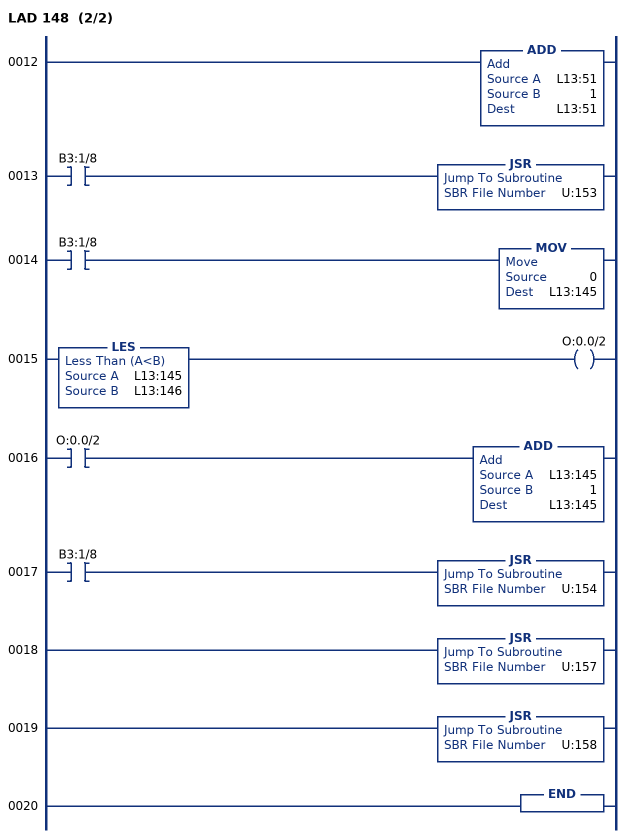
% Rung: 12 %
SOR ADD L13:51 1 L13:51 EOR
% Rung: 13 %
SOR XIC B3:1/8 JSR U:153 EOR
% Rung: 14 %
SOR XIC B3:1/8 MOV 0 L13:145 EOR
% Rung: 15 %
SOR LES L13:145 L13:146 OTE O:0.0/2 EOR
% Rung: 16 %
SOR XIC O:0.0/2 ADD L13:145 1 L13:145 EOR
% Rung: 17 %
SOR XIC B3:1/8 JSR U:154 EOR
% Rung: 18 %
SOR JSR U:157 EOR
% Rung: 19 %
SOR JSR U:158 EOR
% Rung: 20 %
SOR END EOR

LADDER 149
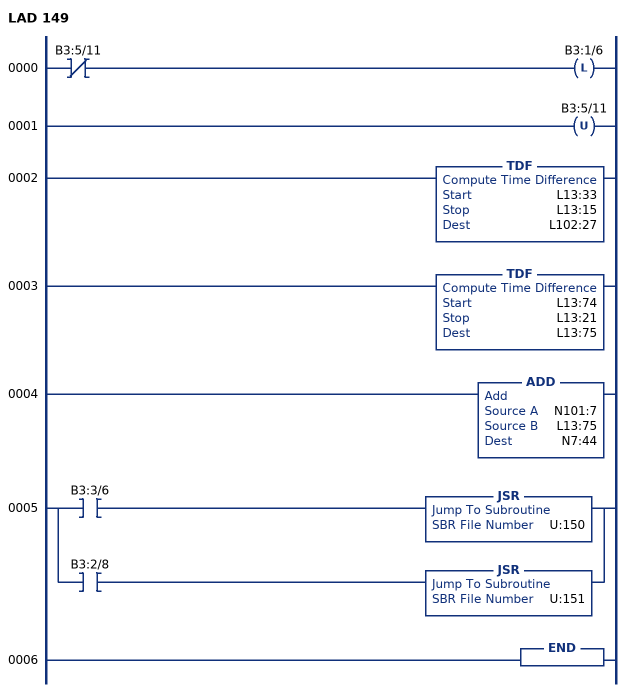
% Rung: 0 %
SOR XIO B3:5/11 OTL B3:1/6 EOR
% Rung: 1 %
SOR OTU B3:5/11 EOR
% Rung: 2 %
SOR TDF L13:33 L13:15 L102:27 EOR
% Rung: 3 %
SOR TDF L13:74 L13:21 L13:75 EOR
% Rung: 4 %
SOR ADD N101:7 L13:75 N7:44 EOR
% Rung: 5 %
SOR BST XIC B3:3/6 JSR U:150 NXB XIC B3:2/8 JSR U:151 BND EOR
% Rung: 6 %
SOR END EOR

LADDER 150
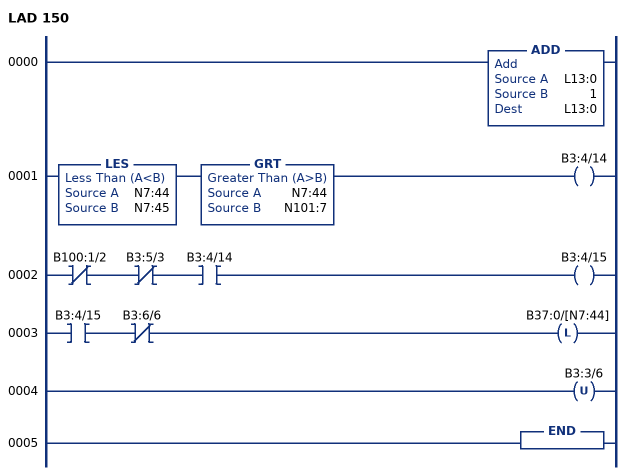
% Rung: 0 %
SOR ADD L13:0 1 L13:0 EOR
% Rung: 1 %
SOR LES N7:44 N7:45 GRT N7:44 N101:7 OTE B3:4/14 EOR
% Rung: 2 %
SOR XIO B100:1/2 XIO B3:5/3 XIC B3:4/14 OTE B3:4/15 EOR
% Rung: 3 %
SOR XIC B3:4/15 XIO B3:6/6 OTL B37:0/[N7:44] EOR
% Rung: 4 %
SOR OTU B3:3/6 EOR
% Rung: 5 %
SOR END EOR

LADDER 151
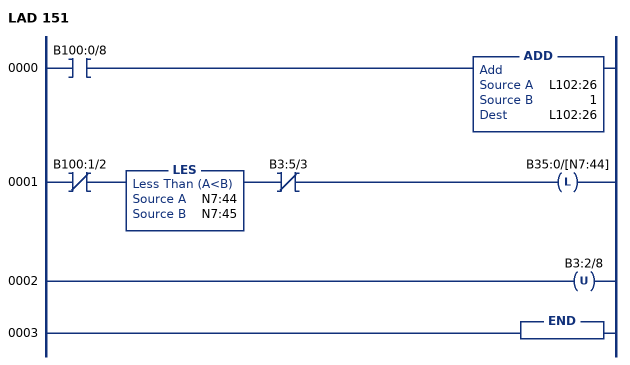
% Rung: 0 %
SOR XIC B100:0/8 ADD L102:26 1 L102:26 EOR
% Rung: 1 %
SOR XIO B100:1/2 LES N7:44 N7:45 XIO B3:5/3 OTL B35:0/[N7:44] EOR
% Rung: 2 %
SOR OTU B3:2/8 EOR
% Rung: 3 %
SOR END EOR

LADDER 152
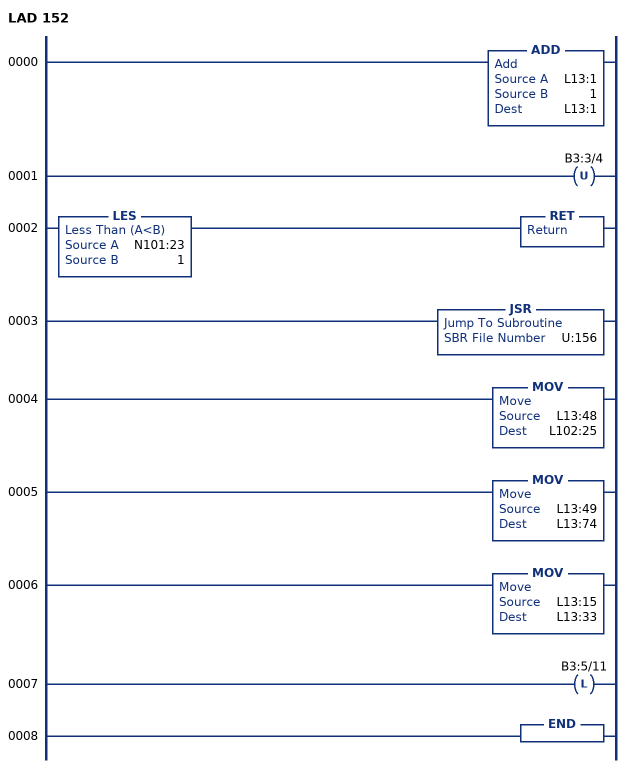
% Rung: 0 %
SOR ADD L13:1 1 L13:1 EOR
% Rung: 1 %
SOR OTU B3:3/4 EOR
% Rung: 2 %
SOR LES N101:23 1 RET EOR
% Rung: 3 %
SOR JSR U:156 EOR
% Rung: 4 %
SOR MOV L13:48 L102:25 EOR
% Rung: 5 %
SOR MOV L13:49 L13:74 EOR
% Rung: 6 %
SOR MOV L13:15 L13:33 EOR
% Rung: 7 %
SOR OTL B3:5/11 EOR
% Rung: 8 %
SOR END EOR

LADDER 153
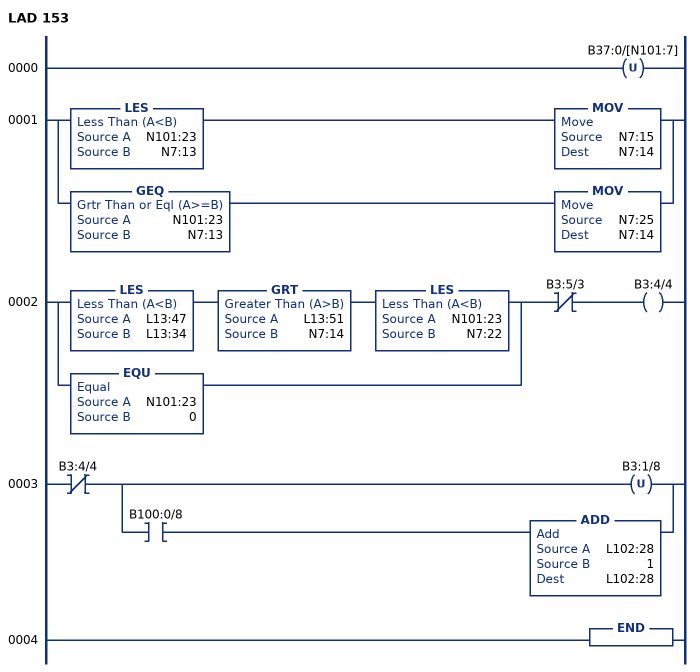
% Rung: 0 %
SOR OTU B37:0/[N101:7] EOR
% Rung: 1 %
SOR BST LES N101:23 N7:13 MOV N7:15 N7:14 NXB GEQ N101:23 N7:13 MOV N7:25 N7:14 BND EOR
% Rung: 2 %
SOR BST LES L13:47 L13:34 GRT L13:51 N7:14 LES N101:23 N7:22 NXB EQU N101:23 0 BND XIO B3:5/3 OTE B3:4/4 EOR
% Rung: 3 %
SOR XIO B3:4/4 BST OTU B3:1/8 NXB XIC B100:0/8 ADD L102:28 1 L102:28 BND EOR
% Rung: 4 %
SOR END EOR

LADDER 154
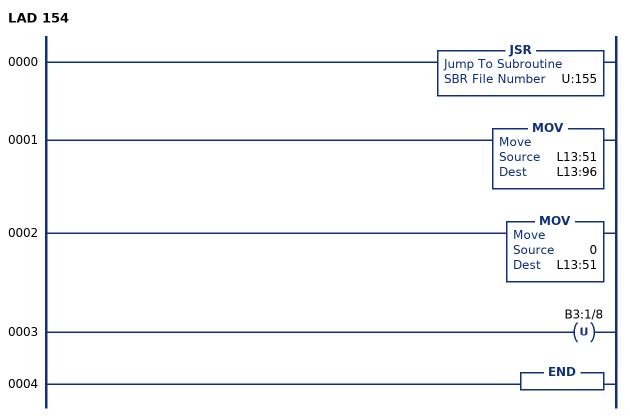
% Rung: 0 %
SOR JSR U:155 EOR
% Rung: 1 %
SOR MOV L13:51 L13:96 EOR
% Rung: 2 %
SOR MOV 0 L13:51 EOR
% Rung: 3 %
SOR OTU B3:1/8 EOR
% Rung: 4 %
SOR END EOR

LADDER 155
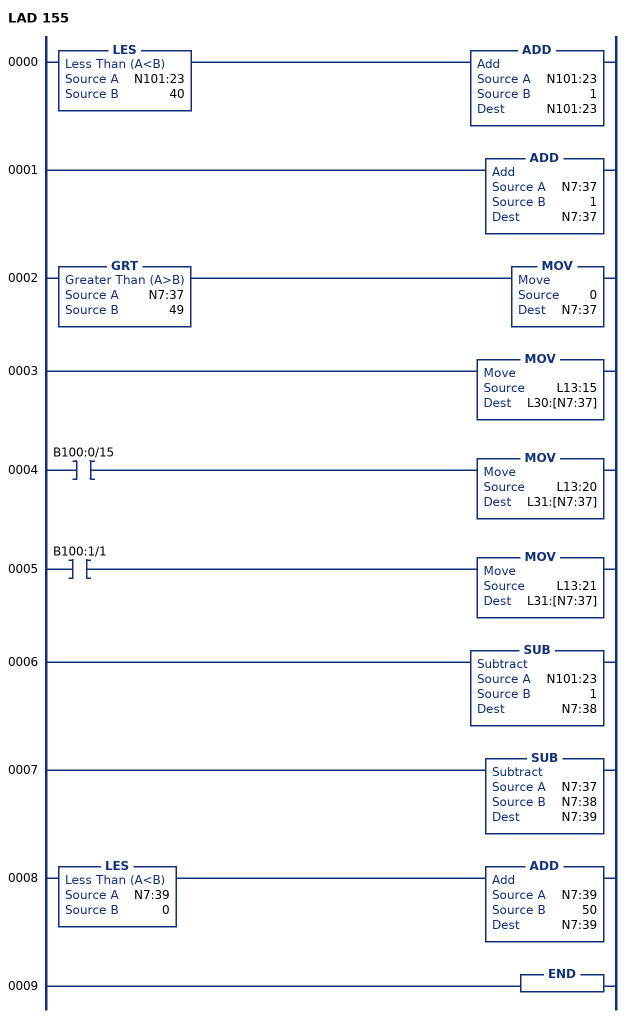
% Rung: 0 %
SOR LES N101:23 40 ADD N101:23 1 N101:23 EOR
% Rung: 1 %
SOR ADD N7:37 1 N7:37 EOR
% Rung: 2 %
SOR GRT N7:37 49 MOV 0 N7:37 EOR
% Rung: 3 %
SOR MOV L13:15 L30:[N7:37] EOR
% Rung: 4 %
SOR XIC B100:0/15 MOV L13:20 L31:[N7:37] EOR
% Rung: 5 %
SOR XIC B100:1/1 MOV L13:21 L31:[N7:37] EOR
% Rung: 6 %
SOR SUB N101:23 1 N7:38 EOR
% Rung: 7 %
SOR SUB N7:37 N7:38 N7:39 EOR
% Rung: 8 %
SOR LES N7:39 0 ADD N7:39 50 N7:39 EOR
% Rung: 9 %
SOR END EOR

LADDER 156
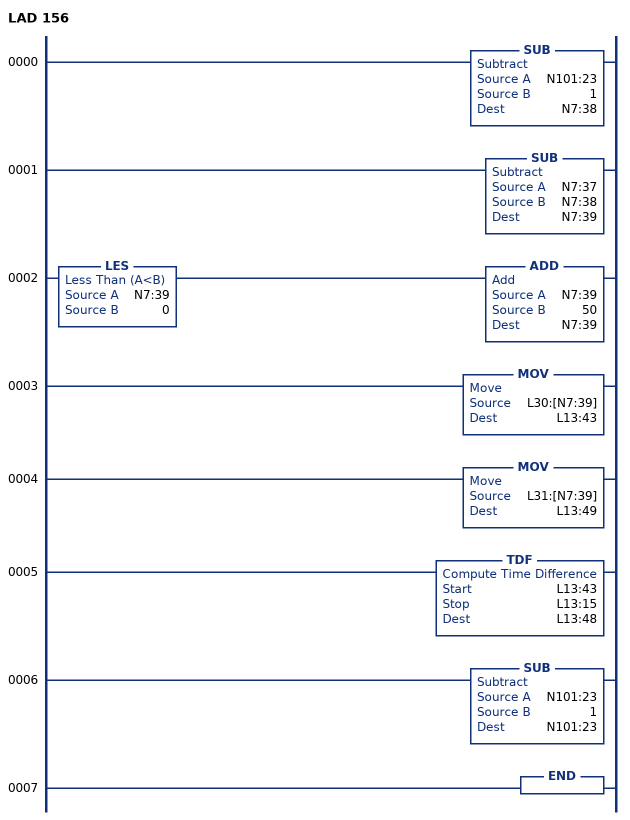
% Rung: 0 %
SOR SUB N101:23 1 N7:38 EOR
% Rung: 1 %
SOR SUB N7:37 N7:38 N7:39 EOR
% Rung: 2 %
SOR LES N7:39 0 ADD N7:39 50 N7:39 EOR
% Rung: 3 %
SOR MOV L30:[N7:39] L13:43 EOR
% Rung: 4 %
SOR MOV L31:[N7:39] L13:49 EOR
% Rung: 5 %
SOR TDF L13:43 L13:15 L13:48 EOR
% Rung: 6 %
SOR SUB N101:23 1 N101:23 EOR
% Rung: 7 %
SOR END EOR

LADDER 157
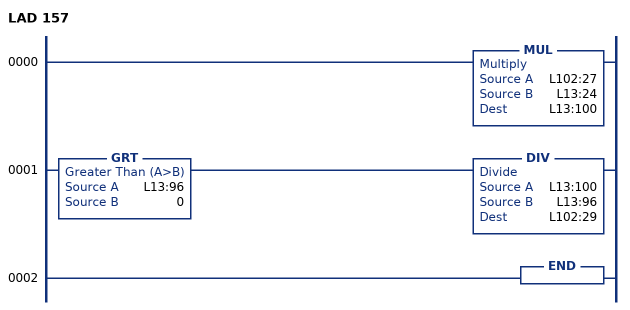
% Rung: 0 %
SOR MUL L102:27 L13:24 L13:100 EOR
% Rung: 1 %
SOR GRT L13:96 0 DIV L13:100 L13:96 L102:29 EOR
% Rung: 2 %
SOR END EOR

LADDER 158
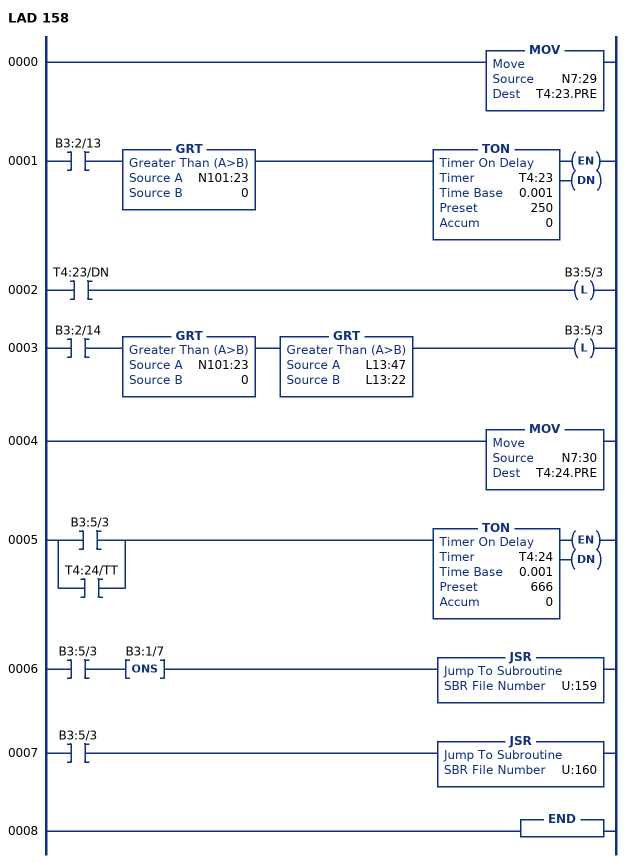
% Rung: 0 %
SOR MOV N7:29 T4:23.PRE EOR
% Rung: 1 %
SOR XIC B3:2/13 GRT N101:23 0 TON T4:23 0.001 250 0 EOR
% Rung: 2 %
SOR XIC T4:23/DN OTL B3:5/3 EOR
% Rung: 3 %
SOR XIC B3:2/14 GRT N101:23 0 GRT L13:47 L13:22 OTL B3:5/3 EOR
% Rung: 4 %
SOR MOV N7:30 T4:24.PRE EOR
% Rung: 5 %
SOR BST XIC B3:5/3 NXB XIC T4:24/TT BND TON T4:24 0.001 666 0 EOR
% Rung: 6 %
SOR XIC B3:5/3 ONS B3:1/7 JSR U:159 EOR
% Rung: 7 %
SOR XIC B3:5/3 JSR U:160 EOR
% Rung: 8 %
SOR END EOR

LADDER 159
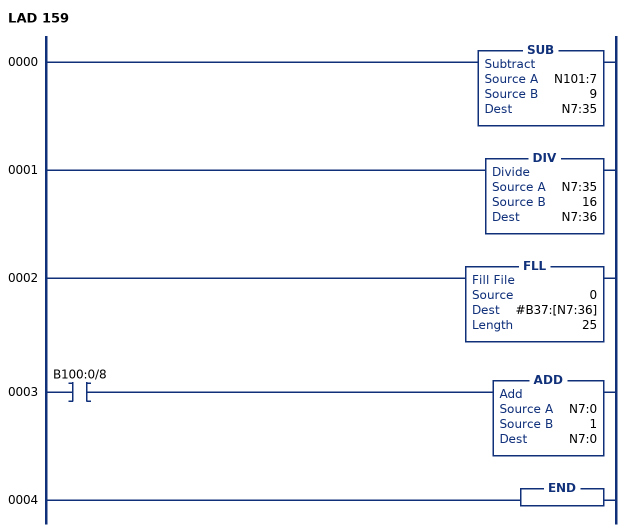
% Rung: 0 %
SOR SUB N101:7 9 N7:35 EOR
% Rung: 1 %
SOR DIV N7:35 16 N7:36 EOR
% Rung: 2 %
SOR FLL 0 #B37:[N7:36] 25 EOR
% Rung: 3 %
SOR XIC B100:0/8 ADD N7:0 1 N7:0 EOR
% Rung: 4 %
SOR END EOR

LADDER 160
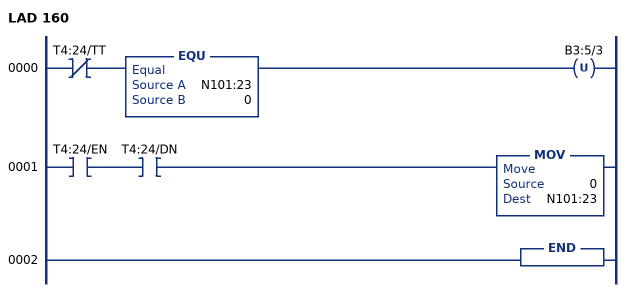
% Rung: 0 %
SOR XIO T4:24/TT EQU N101:23 0 OTU B3:5/3 EOR
% Rung: 1 %
SOR XIC T4:24/EN XIC T4:24/DN MOV 0 N101:23 EOR
% Rung: 2 %
SOR END EOR

LADDER 161
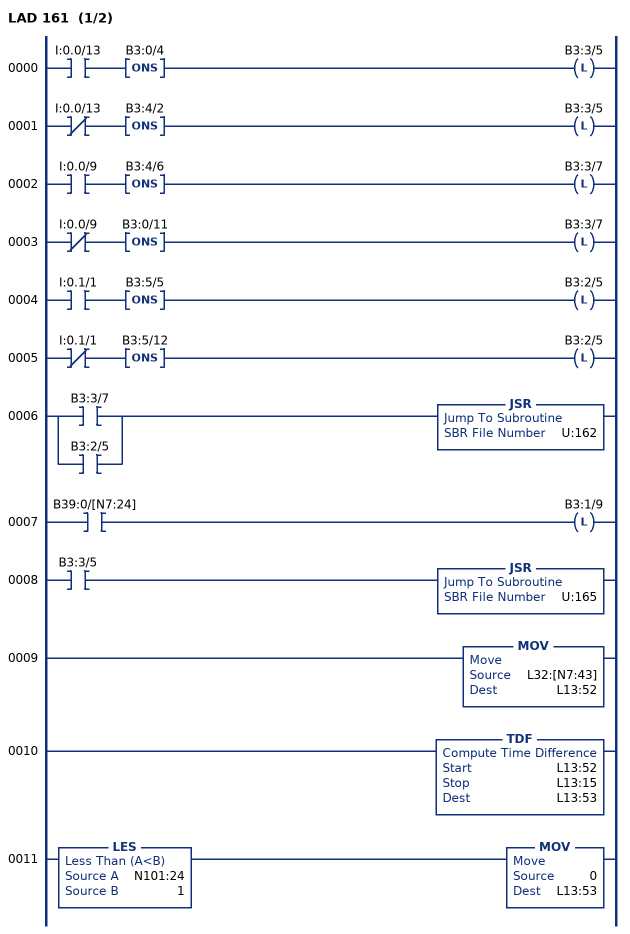
% Rung: 0 %
SOR XIC I:0.0/13 ONS B3:0/4 OTL B3:3/5 EOR
% Rung: 1 %
SOR XIO I:0.0/13 ONS B3:4/2 OTL B3:3/5 EOR
% Rung: 2 %
SOR XIC I:0.0/9 ONS B3:4/6 OTL B3:3/7 EOR
% Rung: 3 %
SOR XIO I:0.0/9 ONS B3:0/11 OTL B3:3/7 EOR
% Rung: 4 %
SOR XIC I:0.1/1 ONS B3:5/5 OTL B3:2/5 EOR
% Rung: 5 %
SOR XIO I:0.1/1 ONS B3:5/12 OTL B3:2/5 EOR
% Rung: 6 %
SOR BST XIC B3:3/7 NXB XIC B3:2/5 BND JSR U:162 EOR
% Rung: 7 %
SOR XIC B39:0/[N7:24] OTL B3:1/9 EOR
% Rung: 8 %
SOR XIC B3:3/5 JSR U:165 EOR
% Rung: 9 %
SOR MOV L32:[N7:43] L13:52 EOR
% Rung: 10 %
SOR TDF L13:52 L13:15 L13:53 EOR
% Rung: 11 %
SOR LES N101:24 1 MOV 0 L13:53 EOR

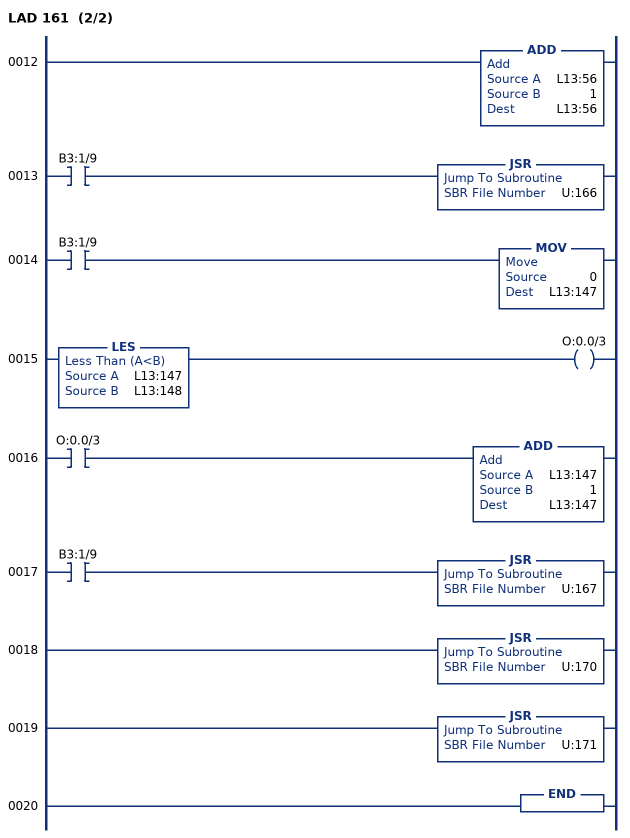
% Rung: 12 %
SOR ADD L13:56 1 L13:56 EOR
% Rung: 13 %
SOR XIC B3:1/9 JSR U:166 EOR
% Rung: 14 %
SOR XIC B3:1/9 MOV 0 L13:147 EOR
% Rung: 15 %
SOR LES L13:147 L13:148 OTE O:0.0/3 EOR
% Rung: 16 %
SOR XIC O:0.0/3 ADD L13:147 1 L13:147 EOR
% Rung: 17 %
SOR XIC B3:1/9 JSR U:167 EOR
% Rung: 18 %
SOR JSR U:170 EOR
% Rung: 19 %
SOR JSR U:171 EOR
% Rung: 20 %
SOR END EOR

LADDER 162
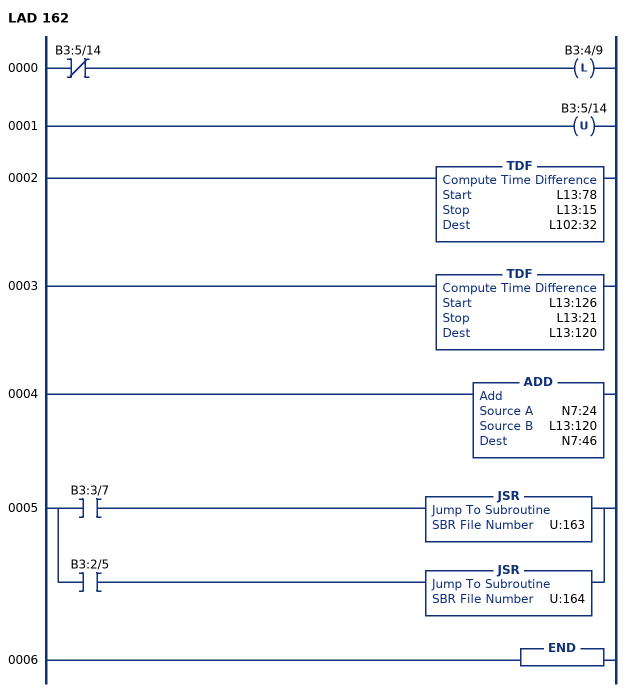
% Rung: 0 %
SOR XIO B3:5/14 OTL B3:4/9 EOR
% Rung: 1 %
SOR OTU B3:5/14 EOR
% Rung: 2 %
SOR TDF L13:78 L13:15 L102:32 EOR
% Rung: 3 %
SOR TDF L13:126 L13:21 L13:120 EOR
% Rung: 4 %
SOR ADD N7:24 L13:120 N7:46 EOR
% Rung: 5 %
SOR BST XIC B3:3/7 JSR U:163 NXB XIC B3:2/5 JSR U:164 BND EOR
% Rung: 6 %
SOR END EOR

LADDER 163
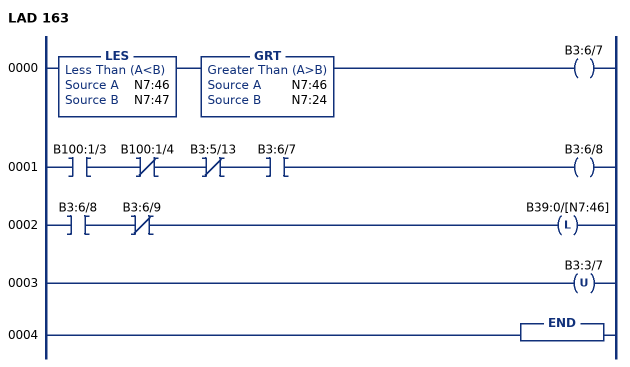
% Rung: 0 %
SOR LES N7:46 N7:47 GRT N7:46 N7:24 OTE B3:6/7 EOR
% Rung: 1 %
SOR XIC B100:1/3 XIO B100:1/4 XIO B3:5/13 XIC B3:6/7 OTE B3:6/8 EOR
% Rung: 2 %
SOR XIC B3:6/8 XIO B3:6/9 OTL B39:0/[N7:46] EOR
% Rung: 3 %
SOR OTU B3:3/7 EOR
% Rung: 4 %
SOR END EOR

LADDER 164
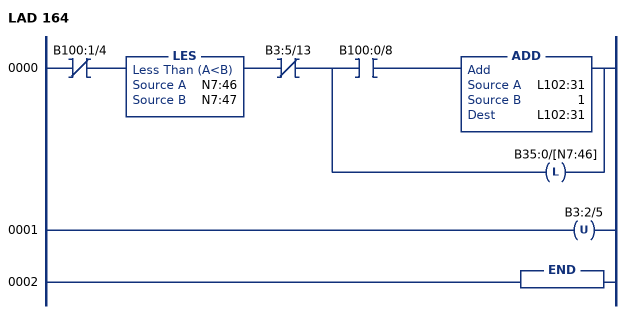
% Rung: 0 %
SOR XIO B100:1/4 LES N7:46 N7:47 XIO B3:5/13 BST XIC B100:0/8 ADD L102:31 1 L102:31 NXB OTL B35:0/[N7:46] BND EOR
% Rung: 1 %
SOR OTU B3:2/5 EOR
% Rung: 2 %
SOR END EOR

LADDER 165
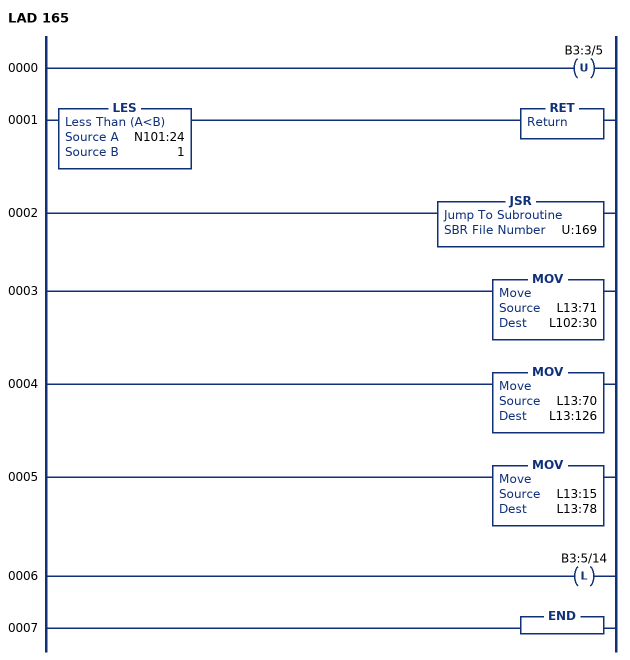
% Rung: 0 %
SOR OTU B3:3/5 EOR
% Rung: 1 %
SOR LES N101:24 1 RET EOR
% Rung: 2 %
SOR JSR U:169 EOR
% Rung: 3 %
SOR MOV L13:71 L102:30 EOR
% Rung: 4 %
SOR MOV L13:70 L13:126 EOR
% Rung: 5 %
SOR MOV L13:15 L13:78 EOR
% Rung: 6 %
SOR OTL B3:5/14 EOR
% Rung: 7 %
SOR END EOR

LADDER 166
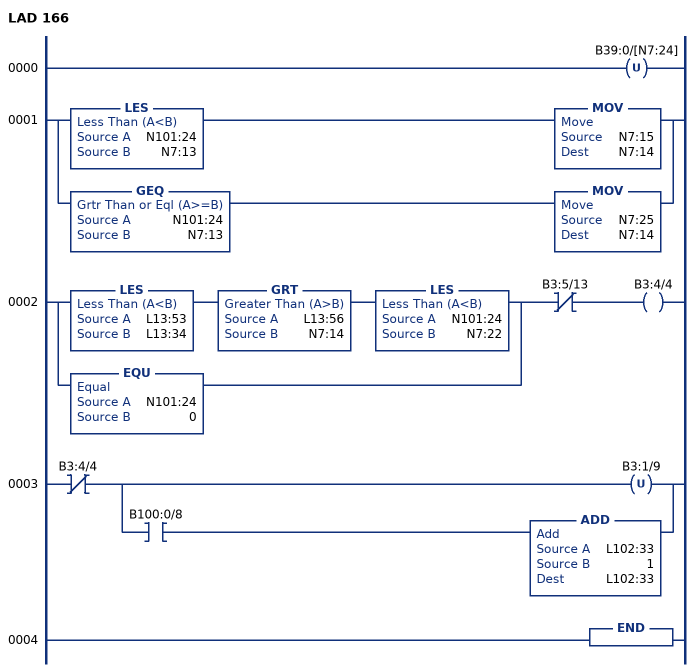
% Rung: 0 %
SOR OTU B39:0/[N7:24] EOR
% Rung: 1 %
SOR BST LES N101:24 N7:13 MOV N7:15 N7:14 NXB GEQ N101:24 N7:13 MOV N7:25 N7:14 BND EOR
% Rung: 2 %
SOR BST LES L13:53 L13:34 GRT L13:56 N7:14 LES N101:24 N7:22 NXB EQU N101:24 0 BND XIO B3:5/13 OTE B3:4/4 EOR
% Rung: 3 %
SOR XIO B3:4/4 BST OTU B3:1/9 NXB XIC B100:0/8 ADD L102:33 1 L102:33 BND EOR
% Rung: 4 %
SOR END EOR

LADDER 167
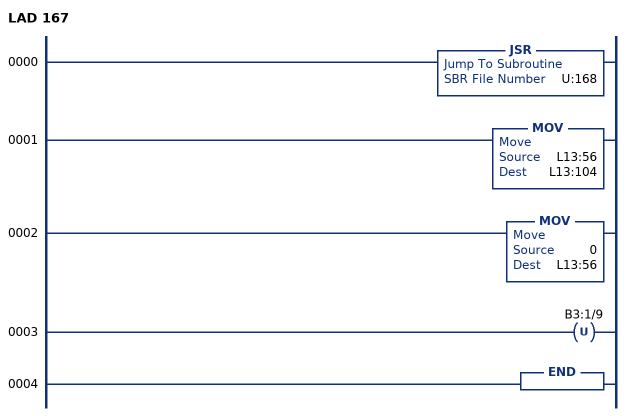
% Rung: 0 %
SOR JSR U:168 EOR
% Rung: 1 %
SOR MOV L13:56 L13:104 EOR
% Rung: 2 %
SOR MOV 0 L13:56 EOR
% Rung: 3 %
SOR OTU B3:1/9 EOR
% Rung: 4 %
SOR END EOR

LADDER 168
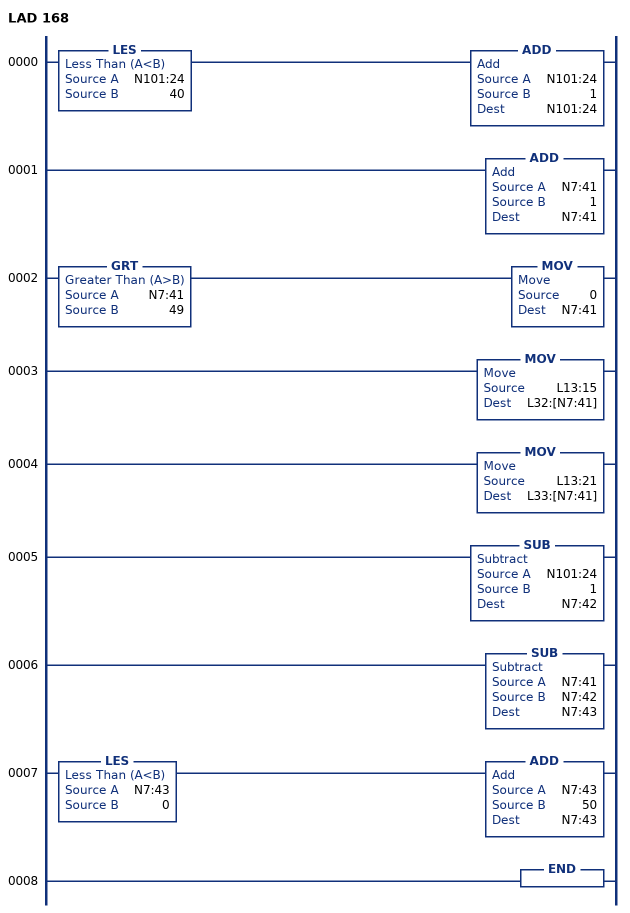
% Rung: 0 %
SOR LES N101:24 40 ADD N101:24 1 N101:24 EOR
% Rung: 1 %
SOR ADD N7:41 1 N7:41 EOR
% Rung: 2 %
SOR GRT N7:41 49 MOV 0 N7:41 EOR
% Rung: 3 %
SOR MOV L13:15 L32:[N7:41] EOR
% Rung: 4 %
SOR MOV L13:21 L33:[N7:41] EOR
% Rung: 5 %
SOR SUB N101:24 1 N7:42 EOR
% Rung: 6 %
SOR SUB N7:41 N7:42 N7:43 EOR
% Rung: 7 %
SOR LES N7:43 0 ADD N7:43 50 N7:43 EOR
% Rung: 8 %
SOR END EOR

LADDER 169
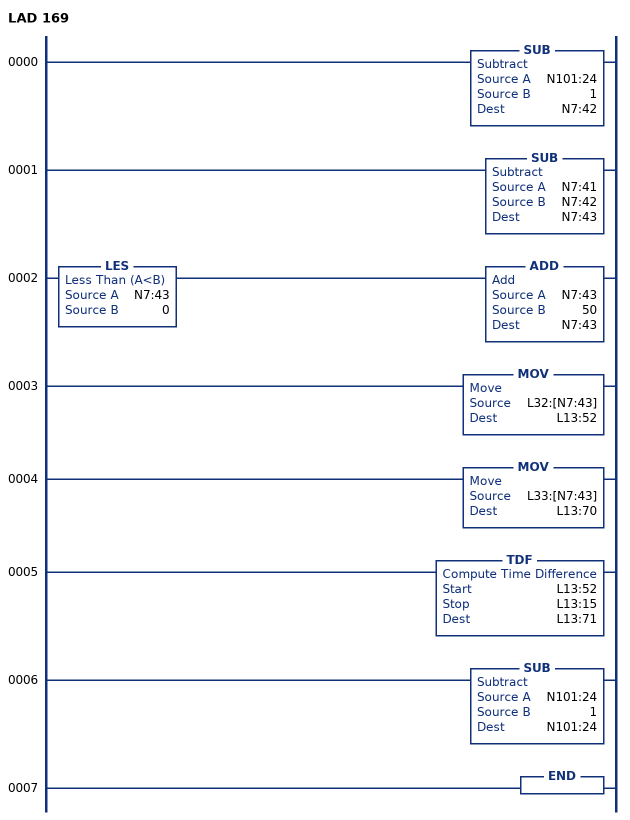
% Rung: 0 %
SOR SUB N101:24 1 N7:42 EOR
% Rung: 1 %
SOR SUB N7:41 N7:42 N7:43 EOR
% Rung: 2 %
SOR LES N7:43 0 ADD N7:43 50 N7:43 EOR
% Rung: 3 %
SOR MOV L32:[N7:43] L13:52 EOR
% Rung: 4 %
SOR MOV L33:[N7:43] L13:70 EOR
% Rung: 5 %
SOR TDF L13:52 L13:15 L13:71 EOR
% Rung: 6 %
SOR SUB N101:24 1 N101:24 EOR
% Rung: 7 %
SOR END EOR

LADDER 170
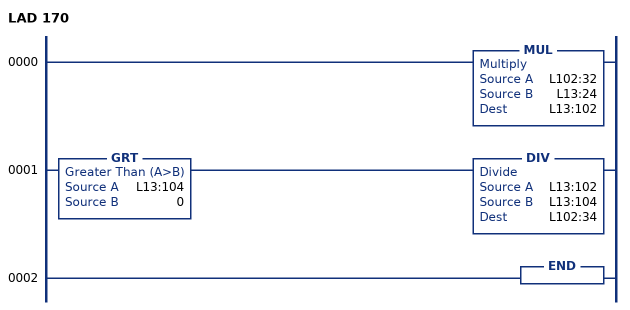
% Rung: 0 %
SOR MUL L102:32 L13:24 L13:102 EOR
% Rung: 1 %
SOR GRT L13:104 0 DIV L13:102 L13:104 L102:34 EOR
% Rung: 2 %
SOR END EOR

LADDER 171
